FUNCTION_BLOCK AxisControl
VAR_INPUT
	//Enable
	McPowerEnable : BOOL;
	//Absolute move
	AbsolutePosition : LREAL;
	ExecuteMoveAbsoluteByManual : BOOL;
	ExecuteMoveAbsoluteByAutomatic : BOOL;
	MoveToBin1 : BOOL;
	MoveToBin2 : BOOL;
	MoveToBin3 : BOOL;
	MoveToBin4 : BOOL;
	//Home move
	ExecuteHomeByManual : BOOL;
	ExecuteHomeByAutomatic : BOOL;
END_VAR
VAR_OUTPUT
	//Position
	ActualPosition : LREAL;
	//Velocity
	ActualVelocity : LREAL;
END_VAR
VAR
	//Power
	McPower : MC_Power;
	McPowerError : BOOL;
	AxisStatus : BOOL;
	//JOG
	McJog : MC_Jog;
	JogForward : BOOL;
	JogBackward : BOOL;

	//Relative
	McMoveRelative : MC_MoveRelative;
	ExecuteRelative : BOOL;
	RelativeDistance : LREAL;
	RelativeVelocity : LREAL;
	//Absolute
	McMoveAbsolute : MC_MoveAbsolute;
	ExecuteAbsolute : BOOL;
	AbsoluteVelocity : LREAL;
	//Velocity
	McMoveVelocity : MC_MoveVelocity;
	ExecuteVelocity : BOOL;
	Velocity : LREAL;
	//Home
	McHome: MC_Home;
	ExecuteHome : BOOL;
	HomeSensor : BOOL;
	//Stop
	McStop : MC_Stop;
	ExecuteStop : BOOL;
	//Halt
	McHalt: MC_Halt;
	ExecuteHalt : BOOL;
END_VAR

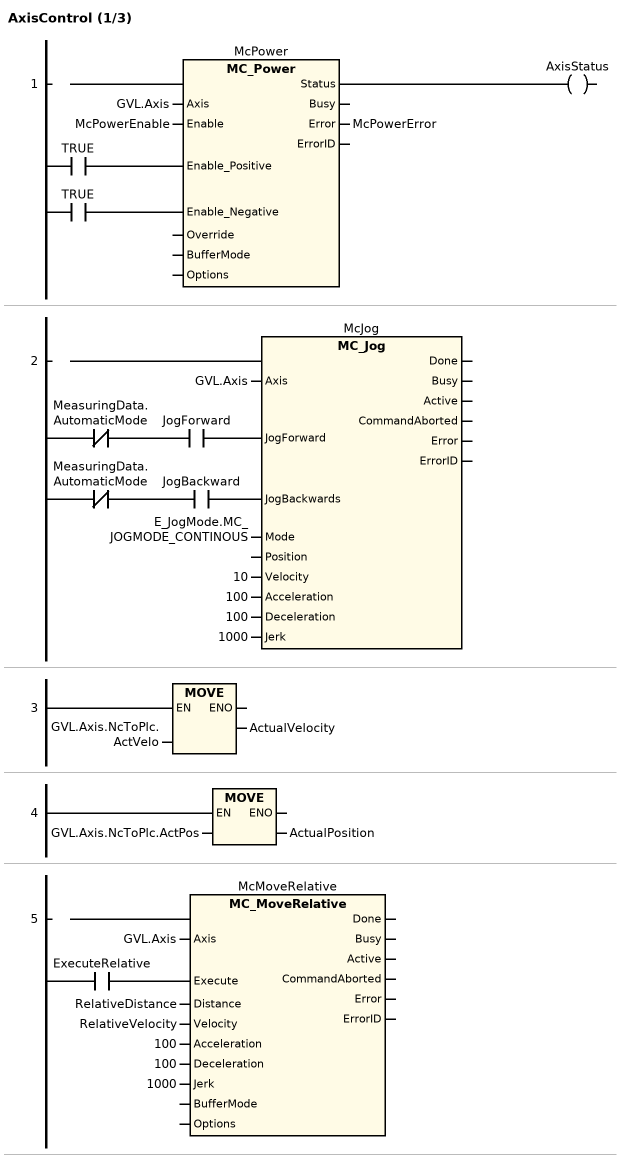
// NETWORK 1
McPower(
    Axis := GVL.Axis,
    Enable := McPowerEnable,
    Enable_Positive := TRUE,
    Enable_Negative := TRUE,
    Error => McPowerError); // MC_Power
AxisStatus := McPower.Status;

// NETWORK 2
McJog(
    Axis := GVL.Axis,
    JogForward := NOT MeasuringData.AutomaticMode AND JogForward,
    JogBackwards := NOT MeasuringData.AutomaticMode AND JogBackward,
    Mode := E_JogMode.MC_JOGMODE_CONTINOUS,
    Velocity := 10,
    Acceleration := 100,
    Deceleration := 100,
    Jerk := 1000); // MC_Jog

// NETWORK 3
ActualVelocity := GVL.Axis.NcToPlc.ActVelo;

// NETWORK 4
ActualPosition := GVL.Axis.NcToPlc.ActPos;

// NETWORK 5
McMoveRelative(
    Axis := GVL.Axis,
    Execute := ExecuteRelative,
    Distance := RelativeDistance,
    Velocity := RelativeVelocity,
    Acceleration := 100,
    Deceleration := 100,
    Jerk := 1000); // MC_MoveRelative

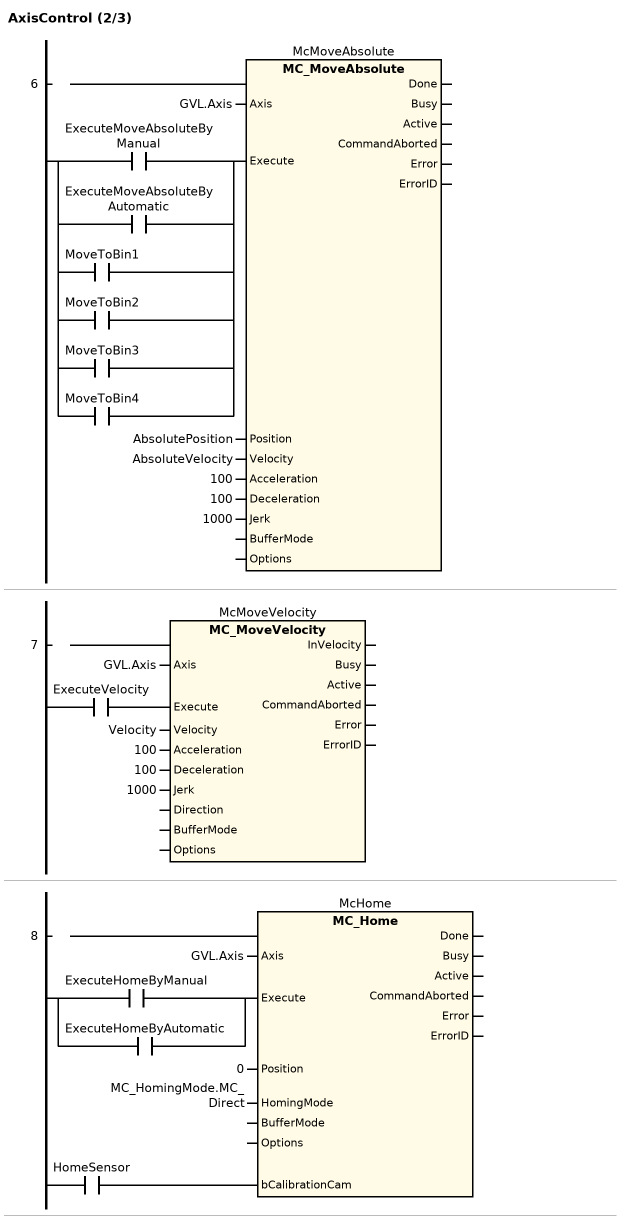
// NETWORK 6
McMoveAbsolute(
    Axis := GVL.Axis,
    Execute := ExecuteMoveAbsoluteByManual OR ExecuteMoveAbsoluteByAutomatic OR MoveToBin1 OR MoveToBin2 OR MoveToBin3 OR MoveToBin4,
    Position := AbsolutePosition,
    Velocity := AbsoluteVelocity,
    Acceleration := 100,
    Deceleration := 100,
    Jerk := 1000); // MC_MoveAbsolute

// NETWORK 7
McMoveVelocity(
    Axis := GVL.Axis,
    Execute := ExecuteVelocity,
    Velocity := Velocity,
    Acceleration := 100,
    Deceleration := 100,
    Jerk := 1000); // MC_MoveVelocity

// NETWORK 8
McHome(
    Axis := GVL.Axis,
    Execute := ExecuteHomeByManual OR ExecuteHomeByAutomatic,
    Position := 0,
    HomingMode := MC_HomingMode.MC_Direct,
    bCalibrationCam := HomeSensor); // MC_Home

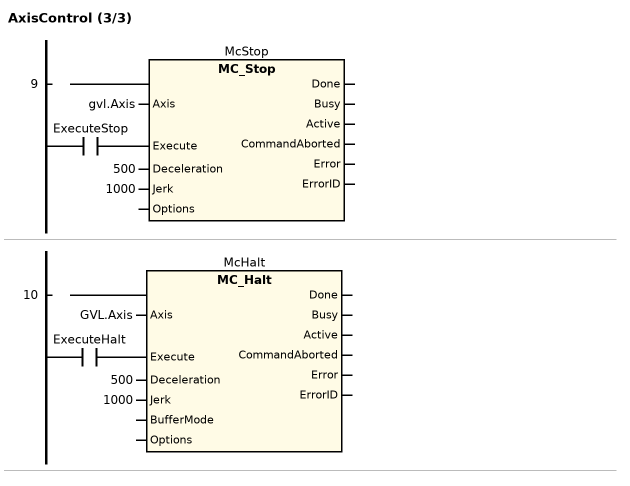
// NETWORK 9
McStop(Axis := gvl.Axis, Execute := ExecuteStop, Deceleration := 500, Jerk := 1000); // MC_Stop

// NETWORK 10
McHalt(Axis := GVL.Axis, Execute := ExecuteHalt, Deceleration := 500, Jerk := 1000); // MC_Halt

END_FUNCTION_BLOCK

(* stored: Version 1.1.0.1, ProductVersion 3.1.4024.13
   POU AxisControl: Id {e3d655ef-40a4-4503-8a77-014b8c965ac4}, SpecialFunc None *)
